Universal Robots PolyScope program: analog_out_test.urp

Program analog_out_test (installation=default directory=/programs createdIn=5.9.5.1031259 lastSavedIn=5.9.5.1031259 robotSerialNumber=20195500451)
Calibrated DH parameters: a=[0.00002, -0.231658, -0.317125, 0.000011, 0.000055, 0]; d=[0.162082, 123.190176, -180.284242, 57.22734, 0.099524, 0.09934]; alpha=[1.569304, 0.00289, 0.004025, 1.569925, -1.569026, 0]; deltaTheta=[0, 0.993923, 4.662183, 0.627072, 0.000001, 0]
Robot Program (runOnlyOnce=false)
  Script: set_analog_outputdomain(0,0)
  count := 0
  Timer (action=Start) variable(name=timer_1)
  Loop Forever
    Script: set_analog_out(0,(sin(timer_1)+1)/2)
